Staubli VAL3: JointTrajPtFMsg.pjx

Parameters version=s7.7.2 stackSize=5000 millimeterUnit=true
Program file=start.pgx
Program file=stop.pgx
Data file=JointTrajPtFMsg.dtx
Type name=Body path=../Body/Body.pjx
Type name=Header path=../Header/Header.pjx
Type name=Prefix path=../Prefix/Prefix.pjx
Type name=JointTrajPtFull path=../JointTrajPtFull/JointTrajPtFull.pjx
